// Mitsubishi GX Works2 project: SEQUENCE_TIMER3   PLC: Q03UDV

PROGRAM MAIN
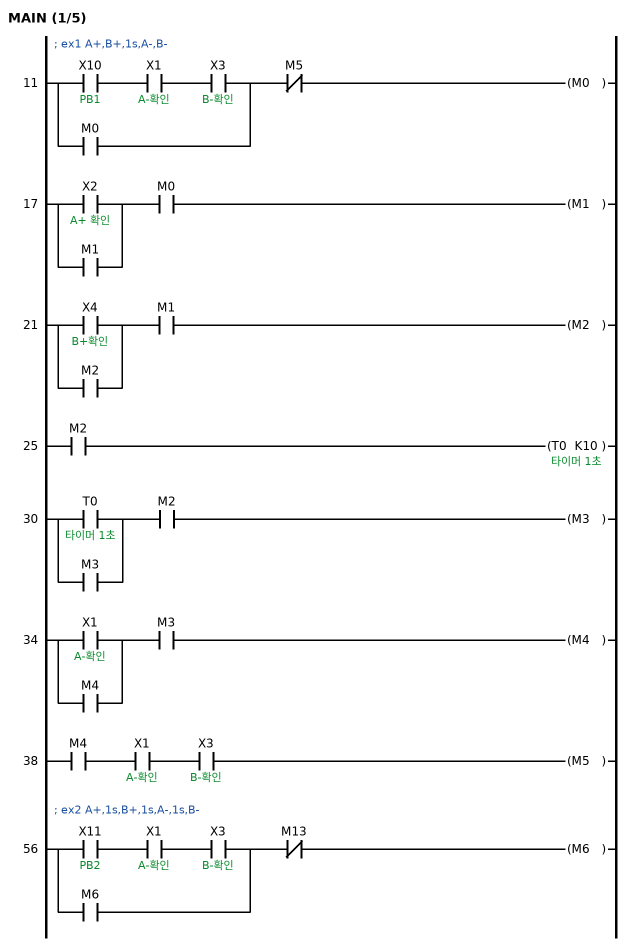
; ex1 A+,B+,1s,A-,B-
11    LD      X10  ; PB1
      AND     X1  ; A-확인
      AND     X3  ; B-확인
      OR      M0
      ANI     M5
      OUT     M0
17    LD      X2  ; A+ 확인
      OR      M1
      AND     M0
      OUT     M1
21    LD      X4  ; B+확인
      OR      M2
      AND     M1
      OUT     M2
25    LD      M2
      OUT     T0 K10  ; 타이머 1초
30    LD      T0  ; 타이머 1초
      OR      M3
      AND     M2
      OUT     M3
34    LD      X1  ; A-확인
      OR      M4
      AND     M3
      OUT     M4
38    LD      M4
      AND     X1  ; A-확인
      AND     X3  ; B-확인
      OUT     M5
; ex2 A+,1s,B+,1s,A-,1s,B-
56    LD      X11  ; PB2
      AND     X1  ; A-확인
      AND     X3  ; B-확인
      OR      M6
      ANI     M13
      OUT     M6
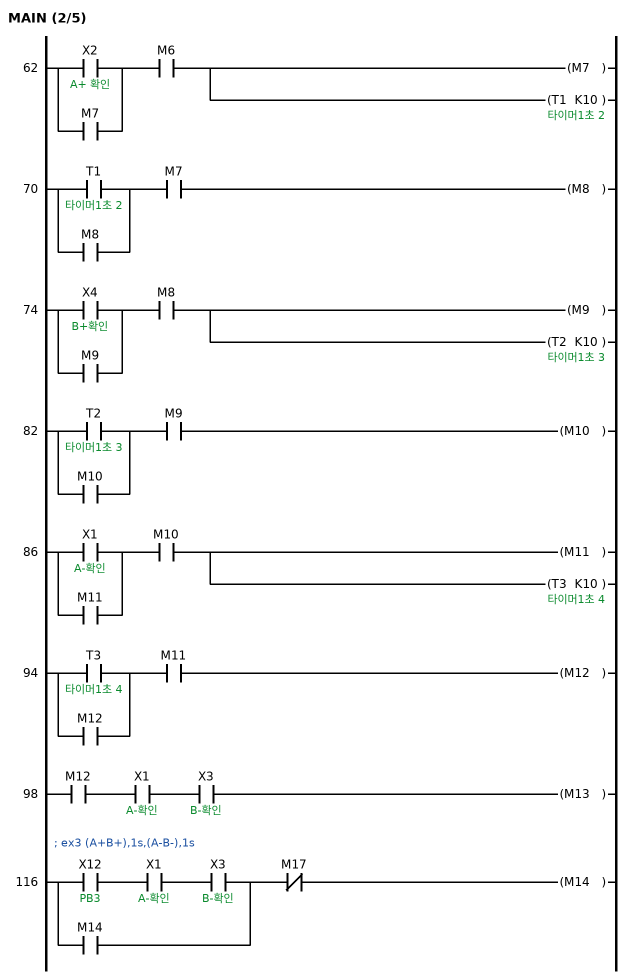
62    LD      X2  ; A+ 확인
      OR      M7
      AND     M6
      OUT     M7
      OUT     T1 K10  ; 타이머1초 2
70    LD      T1  ; 타이머1초 2
      OR      M8
      AND     M7
      OUT     M8
74    LD      X4  ; B+확인
      OR      M9
      AND     M8
      OUT     M9
      OUT     T2 K10  ; 타이머1초 3
82    LD      T2  ; 타이머1초 3
      OR      M10
      AND     M9
      OUT     M10
86    LD      X1  ; A-확인
      OR      M11
      AND     M10
      OUT     M11
      OUT     T3 K10  ; 타이머1초 4
94    LD      T3  ; 타이머1초 4
      OR      M12
      AND     M11
      OUT     M12
98    LD      M12
      AND     X1  ; A-확인
      AND     X3  ; B-확인
      OUT     M13
; ex3 (A+B+),1s,(A-B-),1s
116   LD      X12  ; PB3
      AND     X1  ; A-확인
      AND     X3  ; B-확인
      OR      M14
      ANI     M17
      OUT     M14
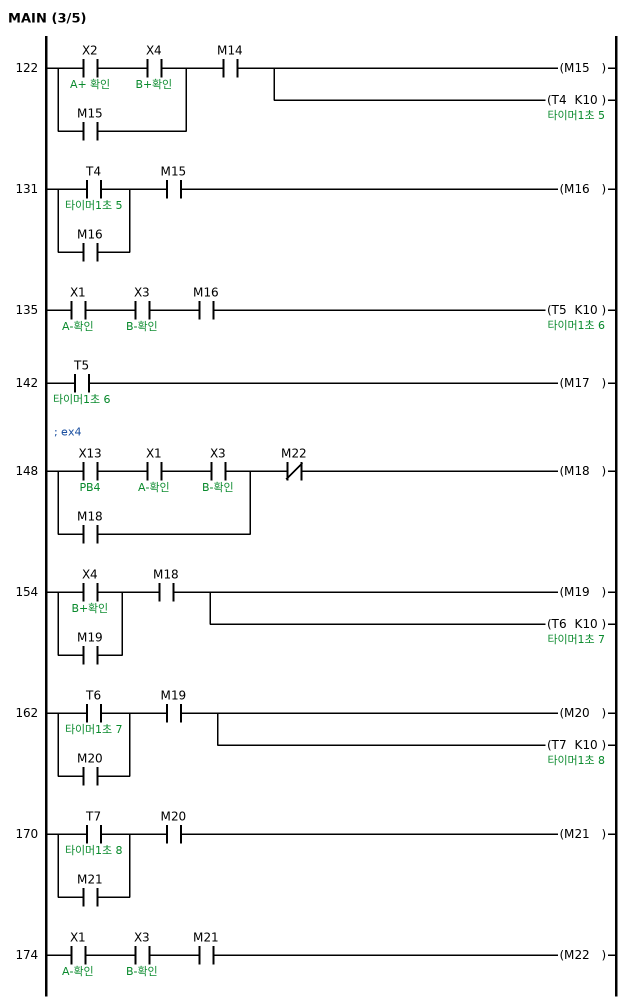
122   LD      X2  ; A+ 확인
      AND     X4  ; B+확인
      OR      M15
      AND     M14
      OUT     M15
      OUT     T4 K10  ; 타이머1초 5
131   LD      T4  ; 타이머1초 5
      OR      M16
      AND     M15
      OUT     M16
135   LD      X1  ; A-확인
      AND     X3  ; B-확인
      AND     M16
      OUT     T5 K10  ; 타이머1초 6
142   LD      T5  ; 타이머1초 6
      OUT     M17
; ex4
148   LD      X13  ; PB4
      AND     X1  ; A-확인
      AND     X3  ; B-확인
      OR      M18
      ANI     M22
      OUT     M18
154   LD      X4  ; B+확인
      OR      M19
      AND     M18
      OUT     M19
      OUT     T6 K10  ; 타이머1초 7
162   LD      T6  ; 타이머1초 7
      OR      M20
      AND     M19
      OUT     M20
      OUT     T7 K10  ; 타이머1초 8
170   LD      T7  ; 타이머1초 8
      OR      M21
      AND     M20
      OUT     M21
174   LD      X1  ; A-확인
      AND     X3  ; B-확인
      AND     M21
      OUT     M22
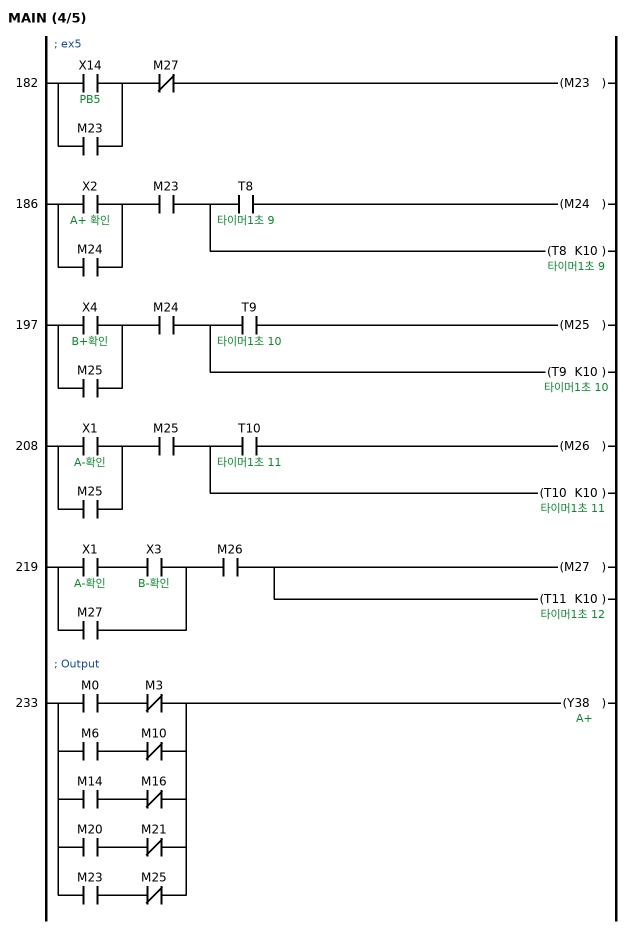
; ex5
182   LD      X14  ; PB5
      OR      M23
      ANI     M27
      OUT     M23
186   LD      X2  ; A+ 확인
      OR      M24
      AND     M23
      MPS
      AND     T8  ; 타이머1초 9
      OUT     M24
      MPP
      OUT     T8 K10  ; 타이머1초 9
197   LD      X4  ; B+확인
      OR      M25
      AND     M24
      MPS
      AND     T9  ; 타이머1초 10
      OUT     M25
      MPP
      OUT     T9 K10  ; 타이머1초 10
208   LD      X1  ; A-확인
      OR      M25
      AND     M25
      MPS
      AND     T10  ; 타이머1초 11
      OUT     M26
      MPP
      OUT     T10 K10  ; 타이머1초 11
219   LD      X1  ; A-확인
      AND     X3  ; B-확인
      OR      M27
      AND     M26
      OUT     M27
      OUT     T11 K10  ; 타이머1초 12
; Output
233   LD      M0
      ANI     M3
      LD      M6
      ANI     M10
      ORB
      LD      M14
      ANI     M16
      ORB
      LD      M20
      ANI     M21
      ORB
      LD      M23
      ANI     M25
      ORB
      OUT     Y38  ; A+
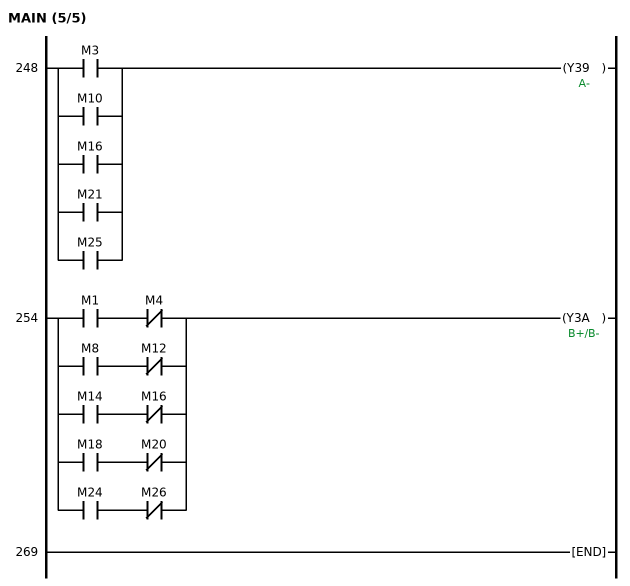
248   LD      M3
      OR      M10
      OR      M16
      OR      M21
      OR      M25
      OUT     Y39  ; A-
254   LD      M1
      ANI     M4
      LD      M8
      ANI     M12
      ORB
      LD      M14
      ANI     M16
      ORB
      LD      M18
      ANI     M20
      ORB
      LD      M24
      ANI     M26
      ORB
      OUT     Y3A  ; B+/B-
269   END
END_PROGRAM
